PROGRAM MAIN
VAR
END_VAR

END_PROGRAM

(* stored: Version 1.1.0.1
   POU MAIN: Id {4d8f841b-6766-4bb2-9c12-099f0a9f66ff} *)
